{attribute 'GeneratedUsingTerminal: EP3162-1002-0017'}
{attribute addProperty BoxType "EP3162-1002-0017"}
{attribute addProperty Id "Digital_outputAT %Q*ARRAY[0..1] OF BOOL2"}
{attribute addProperty CRC "2912513055"}
{attribute addProperty Size "2"}
TYPE DO_Outputs_C0F4C383 EXTENDS OutputBase_10CEE7DE :
STRUCT
	{attribute addProperty Name "Digital_output"}
	Digital_output AT %Q* : ARRAY[0..1] OF BOOL;
END_STRUCT
END_TYPE

(* stored: Version 1.2.0.0, ProductVersion 3.1.4024.9
   DUT DO_Outputs_C0F4C383: Id {92b944d7-b32f-4a9f-b931-af52a10c6105} *)
